Yaskawa INFORM job: ST0RMMYY.JBI

/JOB
//NAME ST0RMMYY
//POS
///NPOS 13,0,0,0
///TOOL 0
///PULSE
C000=-28411,27845,-37313,2831,-2038,2940
C001=-28411,27845,-37313,-4253,146,-448
C002=-28411,27845,-37313,3839,-862,5040
C003=-28411,27845,-37313,-361,-2038,2940
C004=-28411,44357,-37313,-361,-1898,2800
C005=-28411,18101,-37313,-361,-1898,2800
C006=-28411,26165,-37313,-361,-1898,2800
C007=-36619,26165,-37025,-361,-1898,2800
C008=-20635,26165,-37025,-361,-1898,2800
C009=-28843,26165,-37025,2831,-1898,2800
C010=-28843,26165,-37025,-3161,-1898,2800
C011=-28603,26117,-29393,-221,-1898,2800
C012=-28507,26405,-43889,-221,-1898,2800
//INST
///DATE 2014/09/23 21:34
///ATTR 0,0,0,0,0,0,0,0,0,0,0,0,0,0,0,0
///FRAME BASE
NOP
*Y
PAUSE
MOVJ C000 VJ=100.00 CONT
SET B01 0
*M
INC B01
MOVJ C001 VJ=100.00 CONT
MOVJ C002 VJ=100.00 CONT
JUMP *M IF B01<5
MOVJ C003 VJ=100.00 CONT
MOVJ C004 VJ=100.00 CONT
MOVJ C005 VJ=100.00 CONT
MOVJ C006 VJ=100.00 CONT
MOVJ C007 VJ=100.00 CONT
MOVJ C008 VJ=100.00 CONT
MOVJ C009 VJ=100.00 CONT
MOVJ C010 VJ=100.00 CONT
MOVJ C011 VJ=100.00 CONT
MOVJ C012 VJ=100.00 CONT
JUMP *Y
END
